Yaskawa INFORM job: TCP_SHORT_SPIKE.JBI

/JOB
//NAME TCP_SHORT_SPIKE
///FOLDERNAME INNE
//POS
///NPOS 17,17,0,0,0,0
///TOOL 0
///POSTYPE PULSE
///PULSE
C00000=-6252,-3507,65360,7707,108904,32635
C00001=47961,-25136,38328,-379,105651,36537
C00002=100568,-51905,13450,-5853,97534,38171
C00003=168780,-59617,13015,-5805,95821,40923
C00004=-175931,-71226,4547,11199,89426,54882
C00005=-122038,-52934,18016,15115,94974,59536
C00006=-52716,-56516,7003,11411,90818,67922
C00007=-6544,-42730,17642,7627,98410,49309
C00008=21906,-53463,6565,2562,92524,59255
C00009=58850,-68943,-5470,-1969,85973,52576
C00010=133449,-94550,-17329,-7154,72813,48570
C00011=-125723,-113517,-24409,12923,54376,83659
C00012=-24343,-70647,-7159,4275,82402,90666
C00013=-161514,-104836,-19648,12593,66018,63659
C00014=9550,-119911,-28774,1093,36815,84189
C00015=51485,-118556,-28577,-1815,46595,26971
C00016=-93052,-123854,-26359,11664,39579,-57765
BC00000=260759,1064967,688987
BC00001=260759,1064967,688984
BC00002=260759,1064967,688984
BC00003=260759,1064967,688984
BC00004=260759,1064967,688982
BC00005=260759,1064967,688979
BC00006=260759,1064968,688977
BC00007=260759,1064968,688974
BC00008=260759,1064968,688974
BC00009=260759,1064968,688974
BC00010=260759,1064968,688969
BC00011=260759,1064968,688969
BC00012=260759,1064968,688969
BC00013=260759,1064968,688969
BC00014=260759,1064968,688964
BC00015=260759,1064968,688964
BC00016=260759,1064968,688964
//INST
///DATE 2023/10/04 15:12
///ATTR SC,RW
///GROUP1 RB1,BS1
NOP
MOVJ C00000 BC00000 VJ=0.78
MOVJ C00001 BC00001 VJ=0.78
MOVJ C00002 BC00002 VJ=0.78
MOVJ C00003 BC00003 VJ=0.78
MOVJ C00004 BC00004 VJ=0.78
MOVJ C00005 BC00005 VJ=0.78
MOVJ C00006 BC00006 VJ=0.78
MOVJ C00007 BC00007 VJ=0.78
MOVJ C00008 BC00008 VJ=0.78
MOVJ C00009 BC00009 VJ=0.78
MOVJ C00010 BC00010 VJ=0.78
MOVJ C00011 BC00011 VJ=0.78
MOVJ C00012 BC00012 VJ=0.78
MOVJ C00013 BC00013 VJ=0.78
MOVJ C00014 BC00014 VJ=0.78
MOVJ C00015 BC00015 VJ=0.78
MOVJ C00016 BC00016 VJ=0.78
END
